(* IEC 61131-3 sources: Takt/examples/generated/st, 11 files *)

(* ---- batch_cycle.st ---- *)
(*
 * Generated by the Takt compiler (taktc). Target: Structured Text (IEC 61131-3).
 * Do not edit by hand: this file is overwritten on every generation.
 * Takt language version 0.19.0.
 *)

(*
 * Фаза 1: дозирование. Набираем три порции и закрываем клапан.
 *)
FUNCTION_BLOCK BatchCycleDose
VAR_OUTPUT
    is_done : BOOL;
END_VAR
VAR_IN_OUT
    stage : USINT;
END_VAR
VAR
    state : USINT := 0;
    dosed : USINT := 0;
END_VAR
    IF state = 0 THEN (* первый скан *)
        state := 1; (* Fill *)
    END_IF;
    CASE state OF
        1: (* Fill *)
            stage := 1;
            dosed := dosed + 1;
            IF dosed >= 3 THEN
                state := 2; (* Full *)
            END_IF;
        2: (* Full *)
            state := 3; (* END *)
        3: (* END *)
            state := 3;
    END_CASE;
    is_done := state = 3;
END_FUNCTION_BLOCK

(*
 * Фаза 3: слив.
 *)
FUNCTION_BLOCK BatchCycleDrain
VAR_OUTPUT
    is_done : BOOL;
END_VAR
VAR_IN_OUT
    stage : USINT;
END_VAR
VAR
    state : USINT := 0;
    drained : USINT := 0;
END_VAR
    IF state = 0 THEN (* первый скан *)
        state := 2; (* Empty *)
    END_IF;
    CASE state OF
        1: (* Dry *)
            state := 3; (* END *)
        2: (* Empty *)
            stage := 3;
            drained := drained + 1;
            IF drained >= 2 THEN
                state := 1; (* Dry *)
            END_IF;
        3: (* END *)
            state := 3;
    END_CASE;
    is_done := state = 3;
END_FUNCTION_BLOCK

(*
 * Фаза 2: перемешивание.
 *)
FUNCTION_BLOCK BatchCycleMix
VAR_OUTPUT
    is_done : BOOL;
END_VAR
VAR_IN_OUT
    stage : USINT;
END_VAR
VAR
    state : USINT := 0;
    stirred : USINT := 0;
END_VAR
    IF state = 0 THEN (* первый скан *)
        state := 2; (* Stir *)
    END_IF;
    CASE state OF
        1: (* Blended *)
            state := 3; (* END *)
        2: (* Stir *)
            stage := 2;
            stirred := stirred + 1;
            IF stirred >= 2 THEN
                state := 1; (* Blended *)
            END_IF;
        3: (* END *)
            state := 3;
    END_CASE;
    is_done := state = 3;
END_FUNCTION_BLOCK

(*
 * Выходной порт `ready` - наблюдаемая точка завершения цикла: на него смотрит
 * тестбенч цели `sv` (не поднялся - `$error`), причём вместе с порядком фаз.
 * Бит 0 регистра статуса 0x600: цикл завершён. Инициализатор порта задаёт
 * Адрес, а не начальное значение.
 *)
FUNCTION_BLOCK BatchCycle
VAR_OUTPUT
    is_done : BOOL;
    ready : BOOL;
END_VAR
VAR
    state : USINT := 0;
    cycle_dose0 : BatchCycleDose;
    cycle_mix1 : BatchCycleMix;
    cycle_drain2 : BatchCycleDrain;
    cycle_step : USINT;
    stage : USINT := 0;
END_VAR
    IF state = 0 THEN (* первый скан *)
        state := 1; (* Cycle *)
    END_IF;
    CASE state OF
        1: (* Cycle *)
            CASE cycle_step OF
                0:
                    cycle_dose0(stage := stage);
                    IF cycle_dose0.is_done THEN
                        cycle_step := 1;
                    END_IF;
                1:
                    cycle_mix1(stage := stage);
                    IF cycle_mix1.is_done THEN
                        cycle_step := 2;
                    END_IF;
                2:
                    cycle_drain2(stage := stage);
                    IF cycle_drain2.is_done THEN
                        state := 2; (* Done *)
                    END_IF;
            END_CASE;
        2: (* Done *)
            ready := TRUE;
        3: (* END *)
            state := 3;
    END_CASE;
    is_done := state = 3;
END_FUNCTION_BLOCK

(* ---- comprehensive.st ---- *)
(*
 * Generated by the Takt compiler (taktc). Target: Structured Text (IEC 61131-3).
 * Do not edit by hand: this file is overwritten on every generation.
 * Takt language version 0.19.0.
 *)

FUNCTION ComprehensiveController_clamp_temp : USINT
VAR_INPUT
    value : USINT;
END_VAR
VAR CONSTANT
    MAX_TEMP : USINT := 100;
END_VAR
    IF value > MAX_TEMP THEN
        ComprehensiveController_clamp_temp := MAX_TEMP;
        RETURN;
    END_IF;
    ComprehensiveController_clamp_temp := value;
    RETURN;
END_FUNCTION

FUNCTION ComprehensiveController_increment : USINT
VAR_INPUT
    n : USINT;
END_VAR
    ComprehensiveController_increment := n + 1;
    RETURN;
END_FUNCTION

FUNCTION ComprehensiveController_steps_to_limit : USINT
VAR_INPUT
    value : USINT;
END_VAR
VAR
    remaining : USINT;
    v : USINT;
END_VAR
VAR CONSTANT
    HEAT_STEP : USINT := 8;
    MAX_TEMP : USINT := 100;
END_VAR
    remaining := 0;
    v := value;
    WHILE v < MAX_TEMP DO
        v := v + HEAT_STEP;
        remaining := remaining + 1;
    END_WHILE;
    ComprehensiveController_steps_to_limit := remaining;
    RETURN;
END_FUNCTION

FUNCTION ComprehensiveController_steps_to_zero : USINT
VAR_INPUT
    value : USINT;
END_VAR
VAR
    remaining : USINT;
    v : USINT;
END_VAR
VAR CONSTANT
    COOL_STEP : USINT := 3;
END_VAR
    remaining := 0;
    v := value;
    WHILE v > 0 DO
        IF v > COOL_STEP THEN
            v := v - COOL_STEP;
        ELSE
            v := 0;
        END_IF;
        remaining := remaining + 1;
    END_WHILE;
    ComprehensiveController_steps_to_zero := remaining;
    RETURN;
END_FUNCTION

FUNCTION log_count : USINT
VAR_INPUT
    n : USINT;
END_VAR
    log_count := 0;
END_FUNCTION

FUNCTION log_temp : USINT
VAR_INPUT
    value : USINT;
END_VAR
    log_temp := 0;
END_FUNCTION

(*
 * Модель контроллера термоциклирования
 *)
FUNCTION_BLOCK ComprehensiveController
VAR_OUTPUT
    is_done : BOOL;
END_VAR
VAR
    state : USINT := 0;
    i : USINT;
    _st_discard_usint : USINT;
    delta : USINT;
    count : USINT := 0;
    mode : USINT := 0;
    temperature : USINT := 0;
END_VAR
VAR CONSTANT
    Mode_Auto : USINT := 0;
    Mode_Manual : USINT := 1;
    Mode_Emergency : USINT := 2;
    COOL_STEP : USINT := 3;
    HEAT_STEP : USINT := 8;
    MAX_COUNT : USINT := 3;
    MAX_TEMP : USINT := 100;
    WARMUP_TEMP : USINT := 10;
END_VAR
    IF state = 0 THEN (* первый скан *)
        temperature := 0;
        state := 4; (* Idle *)
    END_IF;
    CASE state OF
        1: (* Cooling *)
            i := 0;
            WHILE i < COOL_STEP DO
                IF temperature > 0 THEN
                    temperature := temperature - 1;
                END_IF;
                i := i + 1;
            END_WHILE;
            _st_discard_usint := log_count(ComprehensiveController_steps_to_zero(temperature));
            IF (temperature = 0) AND (count >= MAX_COUNT) THEN
                temperature := 0;
                count := 0;
                state := 2; (* Done *)
            ELSIF (temperature = 0) AND (NOT (count >= MAX_COUNT)) THEN
                temperature := 0;
                state := 4; (* Idle *)
            END_IF;
        2: (* Done *)
            state := 5; (* END *)
        3: (* Heating *)
            temperature := ComprehensiveController_clamp_temp(temperature + HEAT_STEP);
            IF mode = 0 THEN
                _st_discard_usint := log_count(ComprehensiveController_steps_to_limit(temperature));
            ELSIF mode = 1 THEN
                _st_discard_usint := log_temp(temperature);
            ELSE
                mode := Mode_Auto;
            END_IF;
            IF temperature >= MAX_TEMP THEN
                state := 1; (* Cooling *)
            END_IF;
        4: (* Idle *)
            delta := 1;
            temperature := temperature + delta;
            _st_discard_usint := log_temp(temperature);
            IF temperature > WARMUP_TEMP THEN
                count := ComprehensiveController_increment(count);
                state := 3; (* Heating *)
            END_IF;
        5: (* END *)
            state := 5;
    END_CASE;
    is_done := state = 5;
END_FUNCTION_BLOCK

(*
 * Всесторонний пример: демонстрирует возможности языка Takt.
 * Модель - контроллер термоциклирования испытательной камеры: прогреть объект
 * до MAX_TEMP, охладить до нуля, повторить MAX_COUNT раз, завершить работу.
 * Заявленный сценарий: Idle -> Heating -> Cooling -> ... MAX_COUNT раз -> Done;
 * он проверяется прогоном (`takt-sim/tests/sim/examples_scenario_tests.rs`).
 * Использует: переменные, константы, перечисления, внешние функции,
 * условные операторы (if/else), циклы (loop, for, while), вызовы функций,
 * именованные условия (cond), состояния (start/state), оператор match.
 * Перечисление режимов работы
 *)
FUNCTION_BLOCK Comprehensive
VAR_OUTPUT
    is_done : BOOL;
END_VAR
VAR
    state : USINT := 0;
    controller0 : ComprehensiveController;
END_VAR
VAR CONSTANT
    Mode_Auto : USINT := 0;
    Mode_Manual : USINT := 1;
    Mode_Emergency : USINT := 2;
END_VAR
    IF state = 0 THEN (* первый скан *)
        state := 1; (* Entry *)
    END_IF;
    CASE state OF
        1: (* Entry *)
            controller0();
            IF controller0.is_done THEN
                state := 2; (*  *)
            END_IF;
        2: (* END *)
            state := 2;
    END_CASE;
    is_done := state = 2;
END_FUNCTION_BLOCK

(* ---- elevator.st ---- *)
(*
 * Generated by the Takt compiler (taktc). Target: Structured Text (IEC 61131-3).
 * Do not edit by hand: this file is overwritten on every generation.
 * Takt language version 0.19.0.
 *)

FUNCTION door_close : USINT
VAR_INPUT
    unused : USINT;
END_VAR
    door_close := 0;
END_FUNCTION

FUNCTION door_open : USINT
VAR_INPUT
    unused : USINT;
END_VAR
    door_open := 0;
END_FUNCTION

FUNCTION motor_down : USINT
VAR_INPUT
    unused : USINT;
END_VAR
    motor_down := 0;
END_FUNCTION

FUNCTION motor_stop : USINT
VAR_INPUT
    unused : USINT;
END_VAR
    motor_stop := 0;
END_FUNCTION

FUNCTION motor_up : USINT
VAR_INPUT
    unused : USINT;
END_VAR
    motor_up := 0;
END_FUNCTION

FUNCTION read_floor_sensors : USINT
VAR_INPUT
    unused : USINT;
END_VAR
    read_floor_sensors := 0;
END_FUNCTION

FUNCTION scan_cabin_buttons : USINT
VAR_INPUT
    unused : USINT;
END_VAR
    scan_cabin_buttons := 0;
END_FUNCTION

FUNCTION scan_floor_buttons : USINT
VAR_INPUT
    unused : USINT;
END_VAR
    scan_floor_buttons := 0;
END_FUNCTION

(*
 * ══ модель лифта ════════════════════════════════════════════════════════════
 *)
FUNCTION_BLOCK ElevatorEngine
VAR_OUTPUT
    is_done : BOOL;
END_VAR
VAR_IN_OUT
    current_floor : USINT;
    has_call : USINT;
    sensors_cab : USINT;
    target_floor : USINT;
END_VAR
VAR
    state : USINT := 0;
    _st_discard_usint : USINT;
END_VAR
VAR CONSTANT
    Action_Idle : UINT := 670;
    Action_Closing : UINT := 671;
    Floor_Bottom : USINT := 80;
    Floor_Top : USINT := 81;
END_VAR
    IF state = 0 THEN (* первый скан *)
        _st_discard_usint := door_open(0);
        state := 3; (* Idle *)
    END_IF;
    CASE state OF
        1: (* DoorClosing *)
            _st_discard_usint := door_close(0);
            IF ((USINT_TO_BYTE(sensors_cab) AND 16#02) <> 16#00) OR (current_floor = target_floor) THEN
                _st_discard_usint := door_open(0);
                state := 3; (* Idle *)
            ELSIF (NOT ((USINT_TO_BYTE(sensors_cab) AND 16#02) <> 16#00)) AND (current_floor < target_floor) THEN
                state := 5; (* MovingUp *)
            ELSIF (NOT ((USINT_TO_BYTE(sensors_cab) AND 16#02) <> 16#00)) AND (current_floor > target_floor) THEN
                state := 4; (* MovingDown *)
            END_IF;
        2: (* DoorOpening *)
            _st_discard_usint := door_open(0);
            state := 3; (* Idle *)
        3: (* Idle *)
            _st_discard_usint := scan_floor_buttons(0);
            IF (USINT_TO_BYTE(sensors_cab) AND 16#01) <> 16#00 THEN
                _st_discard_usint := scan_cabin_buttons(0);
            END_IF;
            IF (has_call = 1) AND (NOT (current_floor = target_floor)) THEN
                state := 1; (* DoorClosing *)
            END_IF;
        4: (* MovingDown *)
            _st_discard_usint := motor_down(0);
            _st_discard_usint := read_floor_sensors(0);
            _st_discard_usint := scan_floor_buttons(0);
            IF (USINT_TO_BYTE(sensors_cab) AND 16#01) <> 16#00 THEN
                _st_discard_usint := scan_cabin_buttons(0);
            END_IF;
            IF current_floor = target_floor THEN
                _st_discard_usint := motor_stop(0);
                _st_discard_usint := door_open(0);
                has_call := 0;
                state := 2; (* DoorOpening *)
            END_IF;
        5: (* MovingUp *)
            _st_discard_usint := motor_up(0);
            _st_discard_usint := read_floor_sensors(0);
            _st_discard_usint := scan_floor_buttons(0);
            IF (USINT_TO_BYTE(sensors_cab) AND 16#01) <> 16#00 THEN
                _st_discard_usint := scan_cabin_buttons(0);
            END_IF;
            IF current_floor = target_floor THEN
                _st_discard_usint := motor_stop(0);
                _st_discard_usint := door_open(0);
                has_call := 0;
                state := 2; (* DoorOpening *)
            END_IF;
        6: (* END *)
            state := 6;
    END_CASE;
    is_done := state = 6;
END_FUNCTION_BLOCK

(*
 * Схема адресации портов:
 * 0x10000000..0x10000008 - sensors_1..sensors_9
 * 0x10000009             - sensors_cab
 * 0x20000000..0x20000008 - btns_floor_1..btns_floor_9
 * 0x30000000             - btns_cab_lo
 * 0x30000001             - btns_cab_hi
 * ══ порты датчиков положения кабины (1 порт на этаж, 2 бита) ════════════════
 *)
FUNCTION_BLOCK Elevator
VAR_INPUT
    sensors_1 : USINT;
    sensors_2 : USINT;
    sensors_3 : USINT;
    sensors_4 : USINT;
    sensors_5 : USINT;
    sensors_6 : USINT;
    sensors_7 : USINT;
    sensors_8 : USINT;
    sensors_9 : USINT;
    sensors_cab : USINT;
END_VAR
VAR_OUTPUT
    is_done : BOOL;
END_VAR
VAR
    state : USINT := 0;
    engine0 : ElevatorEngine;
    middle_engine1 : ElevatorEngine;
    middle_engine2 : ElevatorEngine;
    middle_engine3 : ElevatorEngine;
    middle_engine4 : ElevatorEngine;
    middle_engine5 : ElevatorEngine;
    middle_engine6 : ElevatorEngine;
    middle_step : USINT;
    current_floor : USINT := 1;
    has_call : USINT := 0;
    target_floor : USINT := 1;
END_VAR
VAR CONSTANT
    Floor_Bottom : USINT := 80;
    Floor_Top : USINT := 81;
END_VAR
    IF state = 0 THEN (* первый скан *)
        state := 2; (* Main *)
    END_IF;
    CASE state OF
        1: (* End *)
            state := 4; (* END *)
        2: (* Main *)
            engine0(current_floor := current_floor, has_call := has_call, sensors_cab := sensors_cab, target_floor := target_floor);
            IF engine0.is_done THEN
                state := 3; (* Middle *)
            END_IF;
        3: (* Middle *)
            CASE middle_step OF
                0:
                    middle_engine1(current_floor := current_floor, has_call := has_call, sensors_cab := sensors_cab, target_floor := target_floor);
                    IF middle_engine1.is_done THEN
                        middle_step := 1;
                    END_IF;
                1:
                    middle_engine2(current_floor := current_floor, has_call := has_call, sensors_cab := sensors_cab, target_floor := target_floor);
                    middle_engine3(current_floor := current_floor, has_call := has_call, sensors_cab := sensors_cab, target_floor := target_floor);
                    IF middle_engine2.is_done AND middle_engine3.is_done THEN
                        middle_step := 2;
                    END_IF;
                2:
                    middle_engine4(current_floor := current_floor, has_call := has_call, sensors_cab := sensors_cab, target_floor := target_floor);
                    IF middle_engine4.is_done THEN
                        middle_step := 3;
                    END_IF;
                3:
                    middle_engine5(current_floor := current_floor, has_call := has_call, sensors_cab := sensors_cab, target_floor := target_floor);
                    IF middle_engine5.is_done THEN
                        middle_step := 4;
                    END_IF;
                4:
                    middle_engine6(current_floor := current_floor, has_call := has_call, sensors_cab := sensors_cab, target_floor := target_floor);
                    IF middle_engine6.is_done THEN
                        state := 1; (* End *)
                    END_IF;
            END_CASE;
        4: (* END *)
            state := 4;
    END_CASE;
    is_done := state = 4;
END_FUNCTION_BLOCK

(* ---- elevator_mini.st ---- *)
(*
 * Generated by the Takt compiler (taktc). Target: Structured Text (IEC 61131-3).
 * Do not edit by hand: this file is overwritten on every generation.
 * Takt language version 0.19.0.
 *)

(*
 * ─── Модель кабины ────────────────────────────────────────────────────────────
 * Idle   - ожидание вызова (door open), обновление этажа, приём кнопок
 * Moving - движение к целевому этажу, постоянное обновление этажа по датчикам
 * AtFloor - прибытие: дверь открыта, ожидаем нажатия DC (закрыть дверь)
 *)
FUNCTION_BLOCK ElevatorMiniCabin
VAR_INPUT
    cabin_button_dc : BOOL;
    cabin_button_f1 : BOOL;
    cabin_button_f2 : BOOL;
    cabin_button_f3 : BOOL;
    cabin_button_f4 : BOOL;
    cabin_button_f5 : BOOL;
    cabin_button_f6 : BOOL;
    cabin_button_f7 : BOOL;
    cabin_button_f8 : BOOL;
    cabin_button_f9 : BOOL;
    floor_button_f1 : BOOL;
    floor_button_f2 : BOOL;
    floor_button_f3 : BOOL;
    floor_button_f4 : BOOL;
    floor_button_f5 : BOOL;
    floor_button_f6 : BOOL;
    floor_button_f7 : BOOL;
    floor_button_f8 : BOOL;
    floor_button_f9 : BOOL;
    floor_sensor_f1_bottom : BOOL;
    floor_sensor_f2_bottom : BOOL;
    floor_sensor_f3_bottom : BOOL;
    floor_sensor_f4_bottom : BOOL;
    floor_sensor_f5_bottom : BOOL;
    floor_sensor_f6_bottom : BOOL;
    floor_sensor_f7_bottom : BOOL;
    floor_sensor_f8_bottom : BOOL;
    floor_sensor_f9_bottom : BOOL;
END_VAR
VAR_OUTPUT
    is_done : BOOL;
    door_open : BOOL;
END_VAR
VAR_IN_OUT
    command : USINT;
    current_floor : USINT;
    target_floor : USINT;
END_VAR
VAR
    state : USINT := 0;
END_VAR
VAR CONSTANT
    Command_Up : USINT := 0;
    Command_Down : USINT := 1;
    Command_Stop : USINT := 2;
END_VAR
    IF state = 0 THEN (* первый скан *)
        command := Command_Stop;
        state := 2; (* Idle *)
    END_IF;
    CASE state OF
        1: (* AtFloor *)
            door_open := TRUE;
            IF cabin_button_dc THEN
                command := Command_Stop;
                state := 2; (* Idle *)
            END_IF;
        2: (* Idle *)
            IF floor_sensor_f1_bottom THEN
                current_floor := 1;
            END_IF;
            IF floor_sensor_f2_bottom THEN
                current_floor := 2;
            END_IF;
            IF floor_sensor_f3_bottom THEN
                current_floor := 3;
            END_IF;
            IF floor_sensor_f4_bottom THEN
                current_floor := 4;
            END_IF;
            IF floor_sensor_f5_bottom THEN
                current_floor := 5;
            END_IF;
            IF floor_sensor_f6_bottom THEN
                current_floor := 6;
            END_IF;
            IF floor_sensor_f7_bottom THEN
                current_floor := 7;
            END_IF;
            IF floor_sensor_f8_bottom THEN
                current_floor := 8;
            END_IF;
            IF floor_sensor_f9_bottom THEN
                current_floor := 9;
            END_IF;
            IF cabin_button_f1 THEN
                target_floor := 1;
            END_IF;
            IF cabin_button_f2 THEN
                target_floor := 2;
            END_IF;
            IF cabin_button_f3 THEN
                target_floor := 3;
            END_IF;
            IF cabin_button_f4 THEN
                target_floor := 4;
            END_IF;
            IF cabin_button_f5 THEN
                target_floor := 5;
            END_IF;
            IF cabin_button_f6 THEN
                target_floor := 6;
            END_IF;
            IF cabin_button_f7 THEN
                target_floor := 7;
            END_IF;
            IF cabin_button_f8 THEN
                target_floor := 8;
            END_IF;
            IF cabin_button_f9 THEN
                target_floor := 9;
            END_IF;
            IF floor_button_f1 THEN
                target_floor := 1;
            END_IF;
            IF floor_button_f2 THEN
                target_floor := 2;
            END_IF;
            IF floor_button_f3 THEN
                target_floor := 3;
            END_IF;
            IF floor_button_f4 THEN
                target_floor := 4;
            END_IF;
            IF floor_button_f5 THEN
                target_floor := 5;
            END_IF;
            IF floor_button_f6 THEN
                target_floor := 6;
            END_IF;
            IF floor_button_f7 THEN
                target_floor := 7;
            END_IF;
            IF floor_button_f8 THEN
                target_floor := 8;
            END_IF;
            IF floor_button_f9 THEN
                target_floor := 9;
            END_IF;
            door_open := TRUE;
            IF target_floor <> 0 THEN
                state := 3; (* Moving *)
            END_IF;
        3: (* Moving *)
            IF floor_sensor_f1_bottom THEN
                current_floor := 1;
            END_IF;
            IF floor_sensor_f2_bottom THEN
                current_floor := 2;
            END_IF;
            IF floor_sensor_f3_bottom THEN
                current_floor := 3;
            END_IF;
            IF floor_sensor_f4_bottom THEN
                current_floor := 4;
            END_IF;
            IF floor_sensor_f5_bottom THEN
                current_floor := 5;
            END_IF;
            IF floor_sensor_f6_bottom THEN
                current_floor := 6;
            END_IF;
            IF floor_sensor_f7_bottom THEN
                current_floor := 7;
            END_IF;
            IF floor_sensor_f8_bottom THEN
                current_floor := 8;
            END_IF;
            IF floor_sensor_f9_bottom THEN
                current_floor := 9;
            END_IF;
            IF target_floor > current_floor THEN
                command := Command_Up;
            END_IF;
            IF target_floor < current_floor THEN
                command := Command_Down;
            END_IF;
            IF target_floor = current_floor THEN
                command := Command_Stop;
                target_floor := 0;
                state := 1; (* AtFloor *)
            END_IF;
        4: (* END *)
            state := 4;
    END_CASE;
    is_done := state = 4;
END_FUNCTION_BLOCK

(*
 * ─── Модель мотора ────────────────────────────────────────────────────────────
 * Простой трёхсостоянный автомат: Idle ↔ Up | Down -> Stop -> Idle.
 * Команда Stop или срабатывание концевого датчика прерывает движение.
 *)
FUNCTION_BLOCK ElevatorMiniMotor
VAR_INPUT
    elevator_motor_sensor_d : BOOL;
    elevator_motor_sensor_u : BOOL;
END_VAR
VAR_OUTPUT
    is_done : BOOL;
    elevator_motor_down : BOOL;
    elevator_motor_stop : BOOL;
    elevator_motor_up : BOOL;
END_VAR
VAR_IN_OUT
    command : USINT;
END_VAR
VAR
    state : USINT := 0;
END_VAR
VAR CONSTANT
    Command_Up : USINT := 0;
    Command_Down : USINT := 1;
    Command_Stop : USINT := 2;
END_VAR
    IF state = 0 THEN (* первый скан *)
        elevator_motor_stop := TRUE;
        state := 2; (* Idle *)
    END_IF;
    CASE state OF
        1: (* Down *)
            elevator_motor_down := TRUE;
            IF (command = Command_Stop) OR elevator_motor_sensor_d THEN
                state := 3; (* Stop *)
            END_IF;
        2: (* Idle *)
            IF command = Command_Up THEN
                state := 4; (* Up *)
            ELSIF command = Command_Down THEN
                state := 1; (* Down *)
            ELSIF command = Command_Stop THEN
                state := 3; (* Stop *)
            END_IF;
        3: (* Stop *)
            elevator_motor_stop := TRUE;
            elevator_motor_stop := TRUE;
            state := 2; (* Idle *)
        4: (* Up *)
            elevator_motor_up := TRUE;
            IF (command = Command_Stop) OR elevator_motor_sensor_u THEN
                state := 3; (* Stop *)
            END_IF;
        5: (* END *)
            state := 5;
    END_CASE;
    is_done := state = 5;
END_FUNCTION_BLOCK

(*
 * Разделяемые переменные (видны обоим авторам):
 * command       : Command  - направление движения, устанавливается Cabin
 * current_floor : u8       - текущий этаж (обновляется по датчикам нижней зоны этажа)
 * target_floor  : u8       - целевой этаж (0 = нет задания)
 *)
FUNCTION_BLOCK ElevatorMini
VAR_OUTPUT
    is_done : BOOL;
END_VAR
VAR
    state : USINT := 0;
    cabin0 : ElevatorMiniCabin;
    motor1 : ElevatorMiniMotor;
    command : USINT := 2;
    current_floor : USINT := 1;
    target_floor : USINT := 0;
END_VAR
VAR CONSTANT
    Command_Up : USINT := 0;
    Command_Down : USINT := 1;
    Command_Stop : USINT := 2;
END_VAR
    IF state = 0 THEN (* первый скан *)
        state := 1; (* Main *)
    END_IF;
    CASE state OF
        1: (* Main *)
            cabin0(command := command, current_floor := current_floor, target_floor := target_floor);
            motor1(command := command);
            IF cabin0.is_done AND motor1.is_done THEN
                state := 2; (*  *)
            END_IF;
        2: (* END *)
            state := 2;
    END_CASE;
    is_done := state = 2;
END_FUNCTION_BLOCK

(* ---- extend_complex.st ---- *)
(*
 * Generated by the Takt compiler (taktc). Target: Structured Text (IEC 61131-3).
 * Do not edit by hand: this file is overwritten on every generation.
 * Takt language version 0.19.0.
 *)

TYPE
    Coord :
    STRUCT
        x : UDINT;
        y : UDINT;
        z : UDINT;
    END_STRUCT;
END_TYPE

FUNCTION has_flag : BOOL
VAR_INPUT
    v : BOOL;
END_VAR
    has_flag := FALSE;
END_FUNCTION

FUNCTION ExtendComplex_is_collected : BOOL
VAR_INPUT
    c : USINT;
    v : USINT;
END_VAR
VAR_IN_OUT
    x : USINT;
END_VAR
    ExtendComplex_is_collected := (((c = 0) AND (v = 1)) OR ((c = 1) AND (v = 2))) OR (((USINT_TO_BYTE(x) AND 16#04) <> 16#00) = 0);
    RETURN;
END_FUNCTION

FUNCTION_BLOCK ExtendComplexA
VAR_OUTPUT
    is_done : BOOL;
END_VAR
VAR
    state : USINT := 0;
END_VAR
VAR CONSTANT
    Constant_X : USINT := 0;
    Constant_Y : USINT := 1;
    Constant_Z : USINT := 2;
    ENABLED : BOOL := TRUE;
END_VAR
    IF state = 0 THEN (* первый скан *)
        state := 1; (* Start *)
    END_IF;
    CASE state OF
        1: (* Start *)
            state := 2; (* END *)
        2: (* END *)
            state := 2;
    END_CASE;
    is_done := state = 2;
END_FUNCTION_BLOCK

FUNCTION_BLOCK ExtendComplexB
VAR_OUTPUT
    is_done : BOOL;
END_VAR
VAR_IN_OUT
    idle : BOOL;
    wait : BOOL;
    work : BOOL;
END_VAR
VAR
    state : USINT := 0;
END_VAR
VAR CONSTANT
    Constant_X : USINT := 0;
    Constant_Y : USINT := 1;
    Constant_Z : USINT := 2;
    ENABLED : BOOL := TRUE;
END_VAR
    IF state = 0 THEN (* первый скан *)
        state := 2; (* Start *)
    END_IF;
    CASE state OF
        1: (* Done *)
            state := 3; (* END *)
        2: (* Start *)
            IF wait THEN
                work := FALSE;
                idle := TRUE;
            ELSE
                idle := FALSE;
                work := TRUE;
            END_IF;
            state := 1; (* Done *)
        3: (* END *)
            state := 3;
    END_CASE;
    is_done := state = 3;
END_FUNCTION_BLOCK

FUNCTION_BLOCK ExtendComplexCC1
VAR_OUTPUT
    is_done : BOOL;
END_VAR
VAR_IN_OUT
    x : USINT;
    y : USINT;
END_VAR
VAR
    state : USINT := 0;
END_VAR
VAR CONSTANT
    Constant_X : USINT := 0;
    Constant_Y : USINT := 1;
    Constant_Z : USINT := 2;
    Point_Global : USINT := 0;
    Point_Local : USINT := 1;
    ENABLED : BOOL := TRUE;
END_VAR
    IF state = 0 THEN (* первый скан *)
        state := 2; (* Start *)
    END_IF;
    CASE state OF
        1: (* End *)
            state := 3; (* END *)
        2: (* Start *)
            IF (ExtendComplex_is_collected(Constant_Y, y) AND ExtendComplex_is_collected(Constant_X, x)) AND has_flag(ENABLED) THEN
                state := 1; (* End *)
            END_IF;
        3: (* END *)
            state := 3;
    END_CASE;
    is_done := state = 3;
END_FUNCTION_BLOCK

FUNCTION_BLOCK ExtendComplexCC2
VAR_OUTPUT
    is_done : BOOL;
END_VAR
VAR
    state : USINT := 0;
END_VAR
VAR CONSTANT
    Constant_X : USINT := 0;
    Constant_Y : USINT := 1;
    Constant_Z : USINT := 2;
    Point_Global : USINT := 0;
    Point_Local : USINT := 1;
    ENABLED : BOOL := TRUE;
END_VAR
    IF state = 0 THEN (* первый скан *)
        state := 1; (* Start *)
    END_IF;
    CASE state OF
        1: (* Start *)
            state := 2; (* END *)
        2: (* END *)
            state := 2;
    END_CASE;
    is_done := state = 2;
END_FUNCTION_BLOCK

FUNCTION_BLOCK ExtendComplexD
VAR_OUTPUT
    is_done : BOOL;
END_VAR
VAR
    state : USINT := 0;
END_VAR
VAR CONSTANT
    Constant_X : USINT := 0;
    Constant_Y : USINT := 1;
    Constant_Z : USINT := 2;
    ENABLED : BOOL := TRUE;
END_VAR
    IF state = 0 THEN (* первый скан *)
        state := 1; (* Start *)
    END_IF;
    CASE state OF
        1: (* Start *)
            state := 2; (* END *)
        2: (* END *)
            state := 2;
    END_CASE;
    is_done := state = 2;
END_FUNCTION_BLOCK

FUNCTION_BLOCK ExtendComplexF
VAR_OUTPUT
    is_done : BOOL;
END_VAR
VAR
    state : USINT := 0;
END_VAR
VAR CONSTANT
    Constant_X : USINT := 0;
    Constant_Y : USINT := 1;
    Constant_Z : USINT := 2;
    ENABLED : BOOL := TRUE;
END_VAR
    IF state = 0 THEN (* первый скан *)
        state := 1; (* Start *)
    END_IF;
    CASE state OF
        1: (* Start *)
            state := 2; (* END *)
        2: (* END *)
            state := 2;
    END_CASE;
    is_done := state = 2;
END_FUNCTION_BLOCK

FUNCTION_BLOCK ExtendComplexC
VAR_OUTPUT
    is_done : BOOL;
END_VAR
VAR_IN_OUT
    x : USINT;
    y : USINT;
END_VAR
VAR
    state : USINT := 0;
    c10 : ExtendComplexCC1;
    c21 : ExtendComplexCC2;
END_VAR
VAR CONSTANT
    Constant_X : USINT := 0;
    Constant_Y : USINT := 1;
    Constant_Z : USINT := 2;
    Point_Global : USINT := 0;
    Point_Local : USINT := 1;
    ENABLED : BOOL := TRUE;
END_VAR
    IF state = 0 THEN (* первый скан *)
        state := 2; (* Start *)
    END_IF;
    CASE state OF
        1: (* End *)
            state := 3; (* END *)
        2: (* Start *)
            c10(x := x, y := y);
            c21();
            IF c10.is_done AND c21.is_done THEN
                state := 1; (* End *)
            END_IF;
        3: (* END *)
            state := 3;
    END_CASE;
    is_done := state = 3;
END_FUNCTION_BLOCK

FUNCTION_BLOCK ExtendComplexE
VAR_OUTPUT
    is_done : BOOL;
END_VAR
VAR
    state : USINT := 0;
    start_d0 : ExtendComplexD;
    start_f1 : ExtendComplexF;
    start_step : USINT;
END_VAR
VAR CONSTANT
    Constant_X : USINT := 0;
    Constant_Y : USINT := 1;
    Constant_Z : USINT := 2;
    ENABLED : BOOL := TRUE;
END_VAR
    IF state = 0 THEN (* первый скан *)
        state := 2; (* Start *)
    END_IF;
    CASE state OF
        1: (* End *)
            state := 3; (* END *)
        2: (* Start *)
            CASE start_step OF
                0:
                    start_d0();
                    IF start_d0.is_done THEN
                        start_step := 1;
                    END_IF;
                1:
                    start_f1();
                    IF start_f1.is_done THEN
                        state := 1; (* End *)
                    END_IF;
            END_CASE;
        3: (* END *)
            state := 3;
    END_CASE;
    is_done := state = 3;
END_FUNCTION_BLOCK

FUNCTION_BLOCK ExtendComplex
VAR_INPUT
    wait : BOOL;
END_VAR
VAR_OUTPUT
    is_done : BOOL;
    idle : BOOL;
    work : BOOL;
END_VAR
VAR
    state : USINT := 0;
    f0 : ExtendComplexF;
    start_a1 : ExtendComplexA;
    start_b2 : ExtendComplexB;
    start_c3 : ExtendComplexC;
    start_d4 : ExtendComplexD;
    start_e5 : ExtendComplexE;
    start_step : USINT;
    x : USINT := 1;
    y : USINT := 2;
END_VAR
VAR CONSTANT
    Constant_X : USINT := 0;
    Constant_Y : USINT := 1;
    Constant_Z : USINT := 2;
    ENABLED : BOOL := TRUE;
END_VAR
    IF state = 0 THEN (* первый скан *)
        state := 2; (* Start *)
    END_IF;
    CASE state OF
        1: (* Next *)
            f0();
            IF f0.is_done THEN
                state := 3; (*  *)
            END_IF;
        2: (* Start *)
            CASE start_step OF
                0:
                    start_a1();
                    IF start_a1.is_done THEN
                        start_step := 1;
                    END_IF;
                1:
                    start_b2(idle := idle, wait := wait, work := work);
                    IF start_b2.is_done THEN
                        start_step := 2;
                    END_IF;
                2:
                    start_c3(x := x, y := y);
                    start_d4();
                    IF start_c3.is_done AND start_d4.is_done THEN
                        start_step := 3;
                    END_IF;
                3:
                    start_e5();
                    IF start_e5.is_done THEN
                        state := 1; (* Next *)
                    END_IF;
            END_CASE;
        3: (* END *)
            state := 3;
    END_CASE;
    is_done := state = 3;
END_FUNCTION_BLOCK

(* ---- float_regulator.st ---- *)
(*
 * Generated by the Takt compiler (taktc). Target: Structured Text (IEC 61131-3).
 * Do not edit by hand: this file is overwritten on every generation.
 * Takt language version 0.19.0.
 *)

(*
 * Обёрнут под-моделью (`start Main = FloatRegulator`): модель без под-моделей не
 * даёт typedef корня в цели `c`. Выходной порт `ready` держит
 * паритет с `regulator.takt` - тот же регулятор, тот же наблюдаемый флаг
 * готовности; проверкой порт здесь не удерживается (в цель `sv` пример без
 * `--float-as-q` не транслируется вовсе - `SV-003`, а контракт сценария
 * проверяет цепочку состояний).
 *)
FUNCTION_BLOCK FloatRegulatorFloatRegulator
VAR_OUTPUT
    is_done : BOOL;
    ready : BOOL;
END_VAR
VAR
    state : USINT := 0;
    half : LREAL := 0.5;
    near : LREAL := 9.5;
    setpoint : LREAL := 10.0;
    value : LREAL := 0.0;
END_VAR
    IF state = 0 THEN (* первый скан *)
        state := 1; (* Adjust *)
    END_IF;
    CASE state OF
        1: (* Adjust *)
            value := value + ((setpoint - value) * half);
            IF value >= near THEN
                state := 3; (* Settled *)
            END_IF;
        2: (* Done *)
            ready := TRUE;
        3: (* Settled *)
            value := setpoint;
            state := 2; (* Done *)
        4: (* END *)
            state := 4;
    END_CASE;
    is_done := state = 4;
END_FUNCTION_BLOCK

(*
 * Обёрнут под-моделью (`start Main = FloatRegulator`): модель без под-моделей не
 * даёт typedef корня в цели `c`. Выходной порт `ready` держит
 * паритет с `regulator.takt` - тот же регулятор, тот же наблюдаемый флаг
 * готовности; проверкой порт здесь не удерживается (в цель `sv` пример без
 * `--float-as-q` не транслируется вовсе - `SV-003`, а контракт сценария
 * проверяет цепочку состояний).
 *)
FUNCTION_BLOCK FloatRegulator
VAR_OUTPUT
    is_done : BOOL;
END_VAR
VAR
    state : USINT := 0;
    float_regulator0 : FloatRegulatorFloatRegulator;
END_VAR
    IF state = 0 THEN (* первый скан *)
        state := 1; (* Main *)
    END_IF;
    CASE state OF
        1: (* Main *)
            float_regulator0();
            IF float_regulator0.is_done THEN
                state := 2; (*  *)
            END_IF;
        2: (* END *)
            state := 2;
    END_CASE;
    is_done := state = 2;
END_FUNCTION_BLOCK

(* ---- pid_heater.st ---- *)
(*
 * Generated by the Takt compiler (taktc). Target: Structured Text (IEC 61131-3).
 * Do not edit by hand: this file is overwritten on every generation.
 * Takt language version 0.19.0.
 *)

TYPE
    PidState :
    STRUCT
        kp : LREAL;
        ki : LREAL;
        kd : LREAL;
        ts : LREAL;
        out_min : LREAL;
        out_max : LREAL;
        i_acc : LREAL;
        err_prev : LREAL;
        output : LREAL;
    END_STRUCT;
END_TYPE

FUNCTION PidHeater_pid_compute : PidState
VAR_INPUT
    p : PidState;
    sp : LREAL;
    pv : LREAL;
END_VAR
VAR
    r : PidState;
    err : LREAL;
    prop : LREAL;
    i_new : LREAL;
    deriv : LREAL;
    raw : LREAL;
END_VAR
    r := p;
    err := sp - pv;
    prop := (p.kp) * err;
    i_new := (p.i_acc) + (((p.ki) * err) * (p.ts));
    deriv := (err - (p.err_prev)) / (p.ts);
    raw := (prop + i_new) + ((p.kd) * deriv);
    IF raw > (p.out_max) THEN
        r.output := p.out_max;
        IF err <= 0.0 THEN
            r.i_acc := i_new;
        END_IF;
    ELSE
        IF raw < (p.out_min) THEN
            r.output := p.out_min;
            IF err >= 0.0 THEN
                r.i_acc := i_new;
            END_IF;
        ELSE
            r.output := raw;
            r.i_acc := i_new;
        END_IF;
    END_IF;
    r.err_prev := err;
    PidHeater_pid_compute := r;
    RETURN;
END_FUNCTION

FUNCTION_BLOCK PidHeaterHeater
VAR_OUTPUT
    is_done : BOOL;
    temperature : LREAL := 0.0;
END_VAR
VAR_IN_OUT
    ambient : LREAL;
    ctrl : LREAL;
    gain : LREAL;
    loss : LREAL;
    meas : LREAL;
    target : LREAL;
END_VAR
VAR
    state : USINT := 0;
    err : LREAL := 0.0;
    loop_pid : PidState := (kp := 0.5, ki := 0.0625, kd := 0.25, ts := 1.0, out_min := 0.0, out_max := 32.0, i_acc := 0.0, err_prev := 0.0, output := 0.0);
    release : LREAL := 38.0;
    setpoint : LREAL := 40.0;
END_VAR
    IF state = 0 THEN (* первый скан *)
        target := setpoint;
        state := 2; (* Heating *)
    END_IF;
    CASE state OF
        1: (* Done *)
            state := 4; (* END *)
        2: (* Heating *)
            (*
             * ─── Шаг закона: операция библиотеки над своим экземпляром ────────
             *)
            loop_pid := PidHeater_pid_compute(loop_pid, target, meas);
            ctrl := loop_pid.output;
            err := target - meas;
            (*
             * ─── Объект: подведённая мощность и потери в среду ────────────────
             *)
            meas := (meas + (gain * ctrl)) - (loss * (meas - ambient));
            temperature := meas;
            IF err <= 0.0 THEN
                ctrl := 0.0;
                state := 3; (* Holding *)
            END_IF;
        3: (* Holding *)
            meas := meas - (loss * (meas - ambient));
            temperature := meas;
            IF meas <= release THEN
                state := 1; (* Done *)
            END_IF;
        4: (* END *)
            state := 4;
    END_CASE;
    is_done := state = 4;
END_FUNCTION_BLOCK

(*
 * Настройка задаётся значениями полей структуры, а не параметрами модели. В
 * этом и разница между регулятором-типом и регулятором-автоматом: контуров
 * столько, сколько объявлено переменных, и каждый несёт свою настройку - а не
 * столько, сколько инстанцировано моделей.
 *)
FUNCTION_BLOCK PidHeater
VAR_OUTPUT
    is_done : BOOL;
END_VAR
VAR
    state : USINT := 0;
    pid_heater_heater0 : PidHeaterHeater;
    pid_heater_heater1 : PidHeaterHeater := (setpoint := 55.0, release := 52.0);
    pid_heater_step : USINT;
    ambient : LREAL := 18.0;
    ctrl : LREAL := 0.0;
    gain : LREAL := 0.5;
    loss : LREAL := 0.05;
    meas : LREAL := 25.0;
    target : LREAL := 80.0;
END_VAR
    IF state = 0 THEN (* первый скан *)
        state := 2; (* PidHeater *)
    END_IF;
    CASE state OF
        1: (* Finished *)
            state := 3; (* END *)
        2: (* PidHeater *)
            CASE pid_heater_step OF
                0:
                    pid_heater_heater0(ambient := ambient, ctrl := ctrl, gain := gain, loss := loss, meas := meas, target := target);
                    IF pid_heater_heater0.is_done THEN
                        pid_heater_step := 1;
                    END_IF;
                1:
                    pid_heater_heater1(ambient := ambient, ctrl := ctrl, gain := gain, loss := loss, meas := meas, target := target);
                    IF pid_heater_heater1.is_done THEN
                        state := 1; (* Finished *)
                    END_IF;
            END_CASE;
        3: (* END *)
            state := 3;
    END_CASE;
    is_done := state = 3;
END_FUNCTION_BLOCK

(* ---- pid_law.st ---- *)
(*
 * Generated by the Takt compiler (taktc). Target: Structured Text (IEC 61131-3).
 * Do not edit by hand: this file is overwritten on every generation.
 * Takt language version 0.19.0.
 *)

TYPE
    (*
     * Файл назван `pid_law.takt`, а не `pid.takt`, намеренно: имя корневой модели
     * берётся из имени файла, и `pid.takt` дал бы корень `PidState` при структуре `PidState`.
     * ─── Состояние одного контура ────────────────────────────────────────────────
     *)
    PidState :
    STRUCT
        kp : LREAL;
        ki : LREAL;
        kd : LREAL;
        ts : LREAL;
        out_min : LREAL;
        out_max : LREAL;
        i_acc : LREAL;
        err_prev : LREAL;
        output : LREAL;
    END_STRUCT;
END_TYPE

FUNCTION PidLaw_pid_compute : PidState
VAR_INPUT
    p : PidState;
    sp : LREAL;
    pv : LREAL;
END_VAR
VAR
    r : PidState;
    err : LREAL;
    prop : LREAL;
    i_new : LREAL;
    deriv : LREAL;
    raw : LREAL;
END_VAR
    r := p;
    err := sp - pv;
    (*
     * Пропорциональная составляющая и новое значение накопителя - пока без
     * ограничений: примем его лишь тогда, когда узнаем, насытился ли выход.
     *)
    prop := (p.kp) * err;
    i_new := (p.i_acc) + (((p.ki) * err) * (p.ts));
    (*
     * Производная - конечная разность назад.
     *)
    deriv := (err - (p.err_prev)) / (p.ts);
    raw := (prop + i_new) + ((p.kd) * deriv);
    IF raw > (p.out_max) THEN
        r.output := p.out_max;
        IF err <= 0.0 THEN
            (*
             * Ошибка толкает выход дальше за верхний предел - накопитель замораживаем.
             *)
            r.i_acc := i_new;
        END_IF;
    ELSE
        IF raw < (p.out_min) THEN
            r.output := p.out_min;
            IF err >= 0.0 THEN
                (*
                 * То же у нижнего предела, зеркально.
                 *)
                r.i_acc := i_new;
            END_IF;
        ELSE
            (*
             * Выход в допустимом диапазоне - накопитель обновляется свободно.
             *)
            r.output := raw;
            r.i_acc := i_new;
        END_IF;
    END_IF;
    r.err_prev := err;
    PidLaw_pid_compute := r;
    RETURN;
END_FUNCTION

FUNCTION PidLaw_pid_init : PidState
VAR_INPUT
    kp : LREAL;
    ki : LREAL;
    kd : LREAL;
    ts : LREAL;
    lo : LREAL;
    hi : LREAL;
END_VAR
VAR
    p : PidState;
END_VAR
    p.kp := 0.0;
    p.ki := 0.0;
    p.kd := 0.0;
    p.ts := 1.0;
    p.out_min := 0.0;
    p.out_max := 0.0;
    p.i_acc := 0.0;
    p.err_prev := 0.0;
    p.output := 0.0;
    p.kp := kp;
    p.ki := ki;
    p.kd := kd;
    p.ts := ts;
    p.out_min := lo;
    p.out_max := hi;
    PidLaw_pid_init := p;
    RETURN;
END_FUNCTION

FUNCTION PidLaw_pid_reset : PidState
VAR_INPUT
    p : PidState;
END_VAR
VAR
    r : PidState;
END_VAR
    r := p;
    r.i_acc := 0.0;
    r.err_prev := 0.0;
    r.output := 0.0;
    PidLaw_pid_reset := r;
    RETURN;
END_FUNCTION

(*
 * Файл назван `pid_law.takt`, а не `pid.takt`, намеренно: имя корневой модели
 * берётся из имени файла, и `pid.takt` дал бы корень `PidState` при структуре `PidState`.
 * ─── Состояние одного контура ────────────────────────────────────────────────
 *)
FUNCTION_BLOCK PidLaw
VAR_OUTPUT
    is_done : BOOL;
END_VAR
VAR
    state : USINT := 0;
    ctrl : LREAL := 0.0;
    hold : BOOL := FALSE;
    loop_pid : PidState := (kp := 3.0, ki := 0.75, kd := 1.5, ts := 0.1, out_min := 0.0, out_max := 100.0, i_acc := 0.0, err_prev := 0.0, output := 0.0);
    meas : LREAL := 25.0;
    target : LREAL := 80.0;
END_VAR
    IF state = 0 THEN (* первый скан *)
        loop_pid := PidLaw_pid_init(3.0, 0.75, 1.5, 0.1, 0.0, 100.0);
        state := 1; (* Run *)
    END_IF;
    CASE state OF
        1: (* Run *)
            loop_pid := PidLaw_pid_compute(loop_pid, target, meas);
            ctrl := loop_pid.output;
            IF hold THEN
                (*
                 * Уставка достигнута - контур перезапускаем, чтобы накопитель не тянул
                 * за собой историю разгона.
                 *)
                loop_pid := PidLaw_pid_reset(loop_pid);
                ctrl := 0.0;
            END_IF;
        2: (* END *)
            state := 2;
    END_CASE;
    is_done := state = 2;
END_FUNCTION_BLOCK

(* ---- pid_regulator.st ---- *)
(*
 * Generated by the Takt compiler (taktc). Target: Structured Text (IEC 61131-3).
 * Do not edit by hand: this file is overwritten on every generation.
 * Takt language version 0.19.0.
 *)

(*
 * Обёрнут под-моделью (цель `c`: typedef корня); порт `ready` - наблюдаемая
 * точка схождения контура, на неё смотрит тестбенч цели `sv` (не поднялся -
 * `$error`). Тела написаны на переменных (не на литералах):
 * литерал `float` в теле дал бы `SV-003` - литералы только в
 * инициализаторах объявлений.
 *)
FUNCTION_BLOCK PidRegulatorPid
VAR_OUTPUT
    is_done : BOOL;
    ready : BOOL;
END_VAR
VAR
    state : USINT := 0;
    ctrl : LREAL := 0.0;
    deriv : LREAL := 0.0;
    eps : LREAL := 0.125;
    err : LREAL := 0.0;
    err_prev : LREAL := 0.0;
    i_acc : LREAL := 0.0;
    imax : LREAL := 32.0;
    kd : LREAL := 0.25;
    ki : LREAL := 0.0625;
    kp : LREAL := 0.5;
    kplant : LREAL := 0.5;
    meas : LREAL := 0.0;
    neg_imax : LREAL := -32.0;
    target : LREAL := 8.0;
END_VAR
    IF state = 0 THEN (* первый скан *)
        state := 1; (* Control *)
    END_IF;
    CASE state OF
        1: (* Control *)
            err := target - meas;
            i_acc := i_acc + err;
            IF i_acc > imax THEN
                i_acc := imax;
            END_IF;
            IF i_acc < neg_imax THEN
                i_acc := neg_imax;
            END_IF;
            deriv := err - err_prev;
            ctrl := ((kp * err) + (ki * i_acc)) + (kd * deriv);
            meas := meas + (kplant * ctrl);
            err_prev := err;
            IF err < eps THEN
                state := 3; (* Settled *)
            END_IF;
        2: (* Done *)
            ready := TRUE;
        3: (* Settled *)
            meas := target;
            state := 2; (* Done *)
        4: (* END *)
            state := 4;
    END_CASE;
    is_done := state = 4;
END_FUNCTION_BLOCK

(*
 * Обёрнут под-моделью (цель `c`: typedef корня); порт `ready` - наблюдаемая
 * точка схождения контура, на неё смотрит тестбенч цели `sv` (не поднялся -
 * `$error`). Тела написаны на переменных (не на литералах):
 * литерал `float` в теле дал бы `SV-003` - литералы только в
 * инициализаторах объявлений.
 *)
FUNCTION_BLOCK PidRegulator
VAR_OUTPUT
    is_done : BOOL;
END_VAR
VAR
    state : USINT := 0;
    pid0 : PidRegulatorPid;
END_VAR
    IF state = 0 THEN (* первый скан *)
        state := 1; (* Main *)
    END_IF;
    CASE state OF
        1: (* Main *)
            pid0();
            IF pid0.is_done THEN
                state := 2; (*  *)
            END_IF;
        2: (* END *)
            state := 2;
    END_CASE;
    is_done := state = 2;
END_FUNCTION_BLOCK

(* ---- regulator.st ---- *)
(*
 * Generated by the Takt compiler (taktc). Target: Structured Text (IEC 61131-3).
 * Do not edit by hand: this file is overwritten on every generation.
 * Takt language version 0.19.0.
 *)

(*
 * Обёрнут под-моделью (`start Main = Regulator`): модель без под-моделей не даёт
 * typedef корня в цели `c`. Выходной порт `ready` - наблюдаемая
 * точка завершения: на него смотрит тестбенч цели `sv` (не поднялся - `$error`),
 * а проверке `sv-mmio` этот пример нужен как единственный, у которого все порты
 * выходные (шине писать некуда - фича). Снимать порт нельзя: оба проверки
 * покраснеют.
 *)
FUNCTION TAKT_Q_FLOORDIV : LINT
VAR_INPUT
    x : LINT;
    d : LINT;
END_VAR
VAR
    q : LINT;
END_VAR
    q := x / d;
    IF (x MOD d <> 0) AND ((x < 0) <> (d < 0)) THEN
        TAKT_Q_FLOORDIV := q - 1;
    ELSE
        TAKT_Q_FLOORDIV := q;
    END_IF;
END_FUNCTION

FUNCTION_BLOCK RegulatorRegulator
VAR_OUTPUT
    is_done : BOOL;
    ready : BOOL;
END_VAR
VAR
    state : USINT := 0;
    half : INT := 128;
    near : INT := 2432;
    setpoint : INT := 2560;
    value : INT := 0;
END_VAR
    IF state = 0 THEN (* первый скан *)
        state := 1; (* Adjust *)
    END_IF;
    CASE state OF
        1: (* Adjust *)
            value := LINT_TO_INT(INT_TO_LINT(value) + INT_TO_LINT(LINT_TO_INT(TAKT_Q_FLOORDIV(INT_TO_LINT((LINT_TO_INT(INT_TO_LINT(setpoint) - INT_TO_LINT(value)))) * INT_TO_LINT(half), 256))));
            IF value >= near THEN
                state := 3; (* Settled *)
            END_IF;
        2: (* Done *)
            ready := TRUE;
        3: (* Settled *)
            value := setpoint;
            state := 2; (* Done *)
        4: (* END *)
            state := 4;
    END_CASE;
    is_done := state = 4;
END_FUNCTION_BLOCK

(*
 * Обёрнут под-моделью (`start Main = Regulator`): модель без под-моделей не даёт
 * typedef корня в цели `c`. Выходной порт `ready` - наблюдаемая
 * точка завершения: на него смотрит тестбенч цели `sv` (не поднялся - `$error`),
 * а проверке `sv-mmio` этот пример нужен как единственный, у которого все порты
 * выходные (шине писать некуда - фича). Снимать порт нельзя: оба проверки
 * покраснеют.
 *)
FUNCTION_BLOCK Regulator
VAR_OUTPUT
    is_done : BOOL;
END_VAR
VAR
    state : USINT := 0;
    regulator0 : RegulatorRegulator;
END_VAR
    IF state = 0 THEN (* первый скан *)
        state := 1; (* Main *)
    END_IF;
    CASE state OF
        1: (* Main *)
            regulator0();
            IF regulator0.is_done THEN
                state := 2; (*  *)
            END_IF;
        2: (* END *)
            state := 2;
    END_CASE;
    is_done := state = 2;
END_FUNCTION_BLOCK

(* ---- stacker.st ---- *)
(*
 * Generated by the Takt compiler (taktc). Target: Structured Text (IEC 61131-3).
 * Do not edit by hand: this file is overwritten on every generation.
 * Takt language version 0.19.0.
 *)

FUNCTION Stacker_travel_time : USINT
VAR_INPUT
    to_stack : USINT;
    to_row : USINT;
    to_section : USINT;
END_VAR
VAR_IN_OUT
    pos_row : USINT;
    pos_section : USINT;
    pos_stack : USINT;
END_VAR
VAR
    ds : USINT;
    dr : USINT;
    dy : USINT;
    t : USINT;
END_VAR
    ds := 0;
    dr := 0;
    dy := 0;
    t := 0;
    IF pos_stack > to_stack THEN
        ds := pos_stack - to_stack;
    ELSE
        ds := to_stack - pos_stack;
    END_IF;
    IF pos_row > to_row THEN
        dr := pos_row - to_row;
    ELSE
        dr := to_row - pos_row;
    END_IF;
    IF pos_section > to_section THEN
        dy := pos_section - to_section;
    ELSE
        dy := to_section - pos_section;
    END_IF;
    t := ds;
    IF dr > t THEN
        t := dr;
    END_IF;
    IF dy > t THEN
        t := dy;
    END_IF;
    Stacker_travel_time := t;
    RETURN;
END_FUNCTION

(*
 * Отслеживает поступление задания от сус и фиксирует принятие на исполнение.
 * Устанавливает cmd_ack=1 в момент приёма, сохраняет параметры в tgt_*.
 * Переходит в TaskActive (busy=1) до момента завершения задания (busy->0).
 *)
FUNCTION_BLOCK StackerCommandReceiver
VAR_OUTPUT
    is_done : BOOL;
END_VAR
VAR_IN_OUT
    busy : BOOL;
    cmd_ack : BOOL;
    eta : USINT;
    sense_battery_low : BOOL;
    task_row_no : USINT;
    task_section_no : USINT;
    task_stack_no : USINT;
    task_type : BOOL;
    task_valid : BOOL;
    tgt_row : USINT;
    tgt_section : USINT;
    tgt_stack : USINT;
    tgt_type : BOOL;
END_VAR
VAR
    state : USINT := 0;
END_VAR
VAR CONSTANT
    CHARGE_ROW : USINT := 0;
    CHARGE_SECTION : USINT := 0;
    CHARGE_STACK : USINT := 0;
    DROPOFF_ROW : USINT := 1;
    DROPOFF_SECTION : USINT := 1;
    DROPOFF_STACK : USINT := 11;
    PICKUP_ROW : USINT := 1;
    PICKUP_SECTION : USINT := 1;
    PICKUP_STACK : USINT := 0;
END_VAR
    IF state = 0 THEN (* первый скан *)
        cmd_ack := FALSE;
        state := 3; (* WaitingForTask *)
    END_IF;
    CASE state OF
        1: (* AcceptingTask *)
            cmd_ack := FALSE;
            state := 2; (* TaskActive *)
        2: (* TaskActive *)
            IF NOT busy THEN
                cmd_ack := FALSE;
                state := 3; (* WaitingForTask *)
            END_IF;
        3: (* WaitingForTask *)
            IF (task_valid AND (NOT busy)) AND (NOT sense_battery_low) THEN
                tgt_stack := task_stack_no;
                tgt_row := task_row_no;
                tgt_section := task_section_no;
                tgt_type := task_type;
                eta := Stacker_travel_time(task_stack_no, task_row_no, task_section_no);
                busy := TRUE;
                cmd_ack := TRUE;
                state := 1; (* AcceptingTask *)
            END_IF;
        4: (* END *)
            state := 4;
    END_CASE;
    is_done := state = 4;
END_FUNCTION_BLOCK

(*
 * Реагирует на запросы от MovementController через lift_request/lift_op.
 * Выдвигает вилы (cmd_fork=1), ожидает целевого состояния груза,
 * убирает вилы и выставляет lift_done. При отмене lift_request немедленно
 * убирает вилы и возвращается в простой.
 *)
FUNCTION_BLOCK StackerLiftController
VAR_OUTPUT
    is_done : BOOL;
END_VAR
VAR_IN_OUT
    cmd_fork : BOOL;
    lift_done : BOOL;
    lift_op : BOOL;
    lift_request : BOOL;
    sense_loaded : BOOL;
END_VAR
VAR
    state : USINT := 0;
END_VAR
VAR CONSTANT
    CHARGE_ROW : USINT := 0;
    CHARGE_SECTION : USINT := 0;
    CHARGE_STACK : USINT := 0;
    DROPOFF_ROW : USINT := 1;
    DROPOFF_SECTION : USINT := 1;
    DROPOFF_STACK : USINT := 11;
    PICKUP_ROW : USINT := 1;
    PICKUP_SECTION : USINT := 1;
    PICKUP_STACK : USINT := 0;
END_VAR
    IF state = 0 THEN (* первый скан *)
        cmd_fork := FALSE;
        state := 2; (* LiftIdle *)
    END_IF;
    CASE state OF
        1: (* LiftDone *)
            IF NOT lift_request THEN
                cmd_fork := FALSE;
                state := 2; (* LiftIdle *)
            END_IF;
        2: (* LiftIdle *)
            IF lift_request THEN
                cmd_fork := TRUE;
                state := 3; (* LiftOperating *)
            END_IF;
        3: (* LiftOperating *)
            IF (lift_request AND (NOT lift_op)) AND sense_loaded THEN
                cmd_fork := FALSE;
                lift_done := TRUE;
                state := 1; (* LiftDone *)
            ELSIF (lift_request AND lift_op) AND (NOT sense_loaded) THEN
                cmd_fork := FALSE;
                lift_done := TRUE;
                state := 1; (* LiftDone *)
            ELSIF NOT lift_request THEN
                cmd_fork := FALSE;
                state := 2; (* LiftIdle *)
            END_IF;
        4: (* END *)
            state := 4;
    END_CASE;
    is_done := state = 4;
END_FUNCTION_BLOCK

(*
 * Управляет целевыми координатами (cmd_target_* ) по трём осям.
 * На каждом этапе, требующем операции вилами, выставляет lift_request и ждёт
 * lift_done от LiftController перед переходом к следующему движению.
 * При разряде батареи прерывает задание и уходит на аварийную зарядку.
 *)
FUNCTION_BLOCK StackerMovementController
VAR_OUTPUT
    is_done : BOOL;
END_VAR
VAR_IN_OUT
    busy : BOOL;
    cmd_ack : BOOL;
    cmd_done : BOOL;
    cmd_target_row : USINT;
    cmd_target_section : USINT;
    cmd_target_stack : USINT;
    lift_done : BOOL;
    lift_op : BOOL;
    lift_request : BOOL;
    pos_row : USINT;
    pos_section : USINT;
    pos_stack : USINT;
    sense_at_charge : BOOL;
    sense_battery_low : BOOL;
    tgt_row : USINT;
    tgt_section : USINT;
    tgt_stack : USINT;
    tgt_type : BOOL;
END_VAR
VAR
    state : USINT := 0;
END_VAR
VAR CONSTANT
    CHARGE_ROW : USINT := 0;
    CHARGE_SECTION : USINT := 0;
    CHARGE_STACK : USINT := 0;
    DROPOFF_ROW : USINT := 1;
    DROPOFF_SECTION : USINT := 1;
    DROPOFF_STACK : USINT := 11;
    PICKUP_ROW : USINT := 1;
    PICKUP_SECTION : USINT := 1;
    PICKUP_STACK : USINT := 0;
END_VAR
    IF state = 0 THEN (* первый скан *)
        cmd_target_stack := CHARGE_STACK;
        cmd_target_row := CHARGE_ROW;
        cmd_target_section := CHARGE_SECTION;
        cmd_done := FALSE;
        state := 3; (* MovementIdle *)
    END_IF;
    CASE state OF
        1: (* DispatchMove *)
            IF NOT tgt_type THEN
                cmd_target_stack := PICKUP_STACK;
                cmd_target_row := PICKUP_ROW;
                cmd_target_section := PICKUP_SECTION;
                state := 6; (* MovingToPickup *)
            ELSIF tgt_type THEN
                lift_request := FALSE;
                lift_done := FALSE;
                cmd_target_stack := tgt_stack;
                cmd_target_row := tgt_row;
                cmd_target_section := tgt_section;
                state := 7; (* MovingToStorage *)
            END_IF;
        2: (* EmergencyCharge *)
            IF sense_at_charge THEN
                cmd_target_stack := CHARGE_STACK;
                cmd_target_row := CHARGE_ROW;
                cmd_target_section := CHARGE_SECTION;
                cmd_done := FALSE;
                state := 3; (* MovementIdle *)
            END_IF;
        3: (* MovementIdle *)
            IF busy AND (NOT sense_battery_low) THEN
                state := 1; (* DispatchMove *)
            END_IF;
        4: (* MovingToCell *)
            IF ((pos_stack = tgt_stack) AND (pos_row = tgt_row)) AND (pos_section = tgt_section) THEN
                lift_request := TRUE;
                lift_op := TRUE;
                state := 9; (* WaitingForkAtCell *)
            ELSIF sense_battery_low THEN
                cmd_target_stack := CHARGE_STACK;
                cmd_target_row := CHARGE_ROW;
                cmd_target_section := CHARGE_SECTION;
                lift_request := FALSE;
                lift_done := FALSE;
                cmd_ack := FALSE;
                cmd_done := FALSE;
                busy := FALSE;
                state := 2; (* EmergencyCharge *)
            END_IF;
        5: (* MovingToDropoff *)
            IF ((pos_stack = DROPOFF_STACK) AND (pos_row = DROPOFF_ROW)) AND (pos_section = DROPOFF_SECTION) THEN
                lift_request := TRUE;
                lift_op := TRUE;
                state := 10; (* WaitingForkAtDropoff *)
            ELSIF sense_battery_low THEN
                cmd_target_stack := CHARGE_STACK;
                cmd_target_row := CHARGE_ROW;
                cmd_target_section := CHARGE_SECTION;
                lift_request := FALSE;
                lift_done := FALSE;
                cmd_ack := FALSE;
                cmd_done := FALSE;
                busy := FALSE;
                state := 2; (* EmergencyCharge *)
            END_IF;
        6: (* MovingToPickup *)
            IF ((pos_stack = PICKUP_STACK) AND (pos_row = PICKUP_ROW)) AND (pos_section = PICKUP_SECTION) THEN
                lift_request := TRUE;
                lift_op := FALSE;
                state := 11; (* WaitingForkAtPickup *)
            ELSIF sense_battery_low THEN
                cmd_target_stack := CHARGE_STACK;
                cmd_target_row := CHARGE_ROW;
                cmd_target_section := CHARGE_SECTION;
                lift_request := FALSE;
                lift_done := FALSE;
                cmd_ack := FALSE;
                cmd_done := FALSE;
                busy := FALSE;
                state := 2; (* EmergencyCharge *)
            END_IF;
        7: (* MovingToStorage *)
            IF ((pos_stack = tgt_stack) AND (pos_row = tgt_row)) AND (pos_section = tgt_section) THEN
                lift_request := TRUE;
                lift_op := FALSE;
                state := 12; (* WaitingForkAtStorage *)
            ELSIF sense_battery_low THEN
                cmd_target_stack := CHARGE_STACK;
                cmd_target_row := CHARGE_ROW;
                cmd_target_section := CHARGE_SECTION;
                lift_request := FALSE;
                lift_done := FALSE;
                cmd_ack := FALSE;
                cmd_done := FALSE;
                busy := FALSE;
                state := 2; (* EmergencyCharge *)
            END_IF;
        8: (* TaskCompleting *)
            cmd_done := FALSE;
            cmd_target_stack := CHARGE_STACK;
            cmd_target_row := CHARGE_ROW;
            cmd_target_section := CHARGE_SECTION;
            cmd_done := FALSE;
            state := 3; (* MovementIdle *)
        9: (* WaitingForkAtCell *)
            IF lift_done THEN
                lift_request := FALSE;
                lift_done := FALSE;
                busy := FALSE;
                cmd_done := TRUE;
                state := 8; (* TaskCompleting *)
            END_IF;
        10: (* WaitingForkAtDropoff *)
            IF lift_done THEN
                lift_request := FALSE;
                lift_done := FALSE;
                busy := FALSE;
                cmd_done := TRUE;
                state := 8; (* TaskCompleting *)
            END_IF;
        11: (* WaitingForkAtPickup *)
            IF lift_done THEN
                lift_request := FALSE;
                lift_done := FALSE;
                cmd_target_stack := tgt_stack;
                cmd_target_row := tgt_row;
                cmd_target_section := tgt_section;
                state := 4; (* MovingToCell *)
            END_IF;
        12: (* WaitingForkAtStorage *)
            IF lift_done THEN
                lift_request := FALSE;
                lift_done := FALSE;
                cmd_target_stack := DROPOFF_STACK;
                cmd_target_row := DROPOFF_ROW;
                cmd_target_section := DROPOFF_SECTION;
                state := 5; (* MovingToDropoff *)
            END_IF;
        13: (* END *)
            state := 13;
    END_CASE;
    is_done := state = 13;
END_FUNCTION_BLOCK

(*
 * Внутренний интерфейс между моделями (координационные переменные):
 * lift_request: MovementController запрашивает операцию вилами
 * lift_op:      тип операции (0=захват, 1=укладка/выдача)
 * lift_done:    LiftController подтверждает завершение операции
 * ─── Константы ────────────────────────────────────────────────────────────────
 *)
FUNCTION_BLOCK Stacker
VAR_INPUT
    pos_row : USINT;
    pos_section : USINT;
    pos_stack : USINT;
    sense_at_charge : BOOL;
    sense_battery_low : BOOL;
    sense_loaded : BOOL;
    task_row_no : USINT;
    task_section_no : USINT;
    task_stack_no : USINT;
    task_type : BOOL;
    task_valid : BOOL;
END_VAR
VAR_OUTPUT
    is_done : BOOL;
    cmd_ack : BOOL;
    cmd_done : BOOL;
    cmd_fork : BOOL;
    cmd_target_row : USINT;
    cmd_target_section : USINT;
    cmd_target_stack : USINT;
END_VAR
VAR
    state : USINT := 0;
    command_receiver0 : StackerCommandReceiver;
    movement_controller1 : StackerMovementController;
    lift_controller2 : StackerLiftController;
    busy : BOOL := FALSE;
    eta : USINT := 0;
    lift_done : BOOL := FALSE;
    lift_op : BOOL := FALSE;
    lift_request : BOOL := FALSE;
    tgt_row : USINT := 0;
    tgt_section : USINT := 0;
    tgt_stack : USINT := 0;
    tgt_type : BOOL := FALSE;
END_VAR
VAR CONSTANT
    CHARGE_ROW : USINT := 0;
    CHARGE_SECTION : USINT := 0;
    CHARGE_STACK : USINT := 0;
    DROPOFF_ROW : USINT := 1;
    DROPOFF_SECTION : USINT := 1;
    DROPOFF_STACK : USINT := 11;
    PICKUP_ROW : USINT := 1;
    PICKUP_SECTION : USINT := 1;
    PICKUP_STACK : USINT := 0;
END_VAR
    IF state = 0 THEN (* первый скан *)
        state := 1; (* Stacker *)
    END_IF;
    CASE state OF
        1: (* Stacker *)
            command_receiver0(busy := busy, cmd_ack := cmd_ack, eta := eta, sense_battery_low := sense_battery_low, task_row_no := task_row_no, task_section_no := task_section_no, task_stack_no := task_stack_no, task_type := task_type, task_valid := task_valid, tgt_row := tgt_row, tgt_section := tgt_section, tgt_stack := tgt_stack, tgt_type := tgt_type);
            movement_controller1(busy := busy, cmd_ack := cmd_ack, cmd_done := cmd_done, cmd_target_row := cmd_target_row, cmd_target_section := cmd_target_section, cmd_target_stack := cmd_target_stack, lift_done := lift_done, lift_op := lift_op, lift_request := lift_request, pos_row := pos_row, pos_section := pos_section, pos_stack := pos_stack, sense_at_charge := sense_at_charge, sense_battery_low := sense_battery_low, tgt_row := tgt_row, tgt_section := tgt_section, tgt_stack := tgt_stack, tgt_type := tgt_type);
            lift_controller2(cmd_fork := cmd_fork, lift_done := lift_done, lift_op := lift_op, lift_request := lift_request, sense_loaded := sense_loaded);
            IF command_receiver0.is_done AND movement_controller1.is_done AND lift_controller2.is_done THEN
                state := 2; (*  *)
            END_IF;
        2: (* END *)
            state := 2;
    END_CASE;
    is_done := state = 2;
END_FUNCTION_BLOCK
